PROGRAM MAIN
VAR
	fbRFID_Reader  : FB_RRU7001;
END_VAR

fbRFID_Reader();

END_PROGRAM

(* stored: Version 1.1.0.1, ProductVersion 3.1.4024.16
   POU MAIN: Id {df3f6be4-87c9-4c81-9aa5-3c217e2e5fbf}, SpecialFunc None *)
